# EPICS StreamDevice protocol: siteApps/danfysikMps9100/danfysikMps9100App/protocol/danfysikMps9100.proto
# Stream Device Protocol for the Danfysik System 9100 power supply
# RS232 (standard version)
#
# Pete Owens 13/5/16
#

OutTerminator = CR;
InTerminator  = LF CR;
ReplyTimeout  = 1000;
ReadTimeout   = 1000;
LockTimeout   = 5000;

adc    { out "AD \$1";      in "%d";          }
wrdac  { out "DA \$1 %d";                     }
rddac  { out "DA \$1";      in "\$1 %d";      }
answer { out "%{NASW|ASW}";                   }
setcmd { out "%{LOC|REM}";                    }
getcmd { out "CMD";         in "%{LOC|REM} "; }
power  { out "%{F|N}";                        }
status { out "S\$1H";       in "%x";          }
first  { out "S1FIRSTH";    in "%x";          }
reset  { out "RS";                            }
setpol { out "PO %{+|-}";                     }
getpol { out "PO";          in "%{+|-}";      }

# just for debugging - actually 2 lines
print  { out "PRINT";       in "%39c" ;       }
